// TIA Portal V18 export
DATA_BLOCK "BoilerOnOffSettings"   // DB1017
{ S7_Optimized_Access := 'FALSE' }
VERSION : 0.1
// stored: AutoNumber false, DBAccessibleFromOPCUA true, IsOnlyStoredInLoadMemory false, IsWriteProtectedInAS false
   VAR
      Boiler { S7_SetPoint := 'True'} : "UDT_BoilersOnOffSettings";
   END_VAR
BEGIN
   Boiler.PLCModeSelection.cPreselectedOpModePLC := 16#3;
   Boiler.PLCModeSelection.cActualOpModePLC := 16#3;
END_DATA_BLOCK
